FUNCTION_BLOCK "G280M_Code"
TITLE =G280M CHAIN CONVEYOR 9001 KILN 1
//COPYRIGHT:    (C) 2009  BUHLER AG, CH-9240 UZWIL, SWITZERLAND
//
//PRODUCT:      WinCoS_BIW01_09
//
//TITLE:        CHAIN CONVEYOR 9001 KILN 1
//                Machine group control
//                Maschinengruppensteuerung
//
//--------------------------------------------------------------------------------
//
//IDENT:        AUTHOR:             DEPT:                              DATE:
//
//P01_FB380.1.0 K.Renz              CSB41                              08.Jun.2010
//             1st Release
//
//--------------------------------------------------------------------------------
//
//PURPOSE:
//
//MANUAL :
//
//RESTRICTIONS:
//
//--------------------------------------------------------------------------------
AUTHOR : KR
FAMILY : USW
VERSION : 9.9


VAR
  Gr : "GCS7_GrpCtrlSub";	//Standard interface to group
  InOutValue1 : DINT ;	//Data for user
  InOutValue2 : DINT ;	//Data for user
  OutWayConflict : BOOL ;	//Data for user
  OutSelectionOk : BOOL ;	//Data for user
  CmdNewValue : BOOL ;	//Data for user
  CmdNewJob : BOOL ;	//Data for user
  OutCodeOK : BOOL ;	//Data for user
  InEndOfJob : BOOL ;	//Data for user
  staWayOk : BOOL ;	//Data for user
  EdgeStartRelease : BOOL ;	//Data for user
  USW8 : BOOL ;	//Data for user
  USW9 : BOOL ;	//Data for user
  USW10 : BOOL ;	//Data for user
  USW11 : BOOL ;	//Data for user
  USW12 : BOOL ;	//Data for user
  USW13 : BOOL ;	//Data for user
  USW14 : BOOL ;	//Data for user
  USW15 : BOOL ;	//Data for user
  A_3922_BZS04 : "GCS7_E_DigInput";	// DigInpCont
  A_3922_BZS05 : "GCS7_E_DigInput";	// DigInpCont
  A_3922_MXZ01 : "GCS7_E_Motor";	// Motor
  A_3921_MXZ01MA : "A_3921_MXZ01MA_Code";	// Motor+6DI
END_VAR
VAR_TEMP
  tmpEnable : BOOL ;
  tmpFlag : BOOL ;
  tmpCmdNext : BOOL ;
  tmpLocal : BOOL ;
  tmpAspOk : BOOL ;
  tmpHWStop : BOOL ;
  tmpInstanzDBNo : INT ;
END_VAR
BEGIN
NETWORK
TITLE =



NETWORK
TITLE =Read command from group control
//Parameter
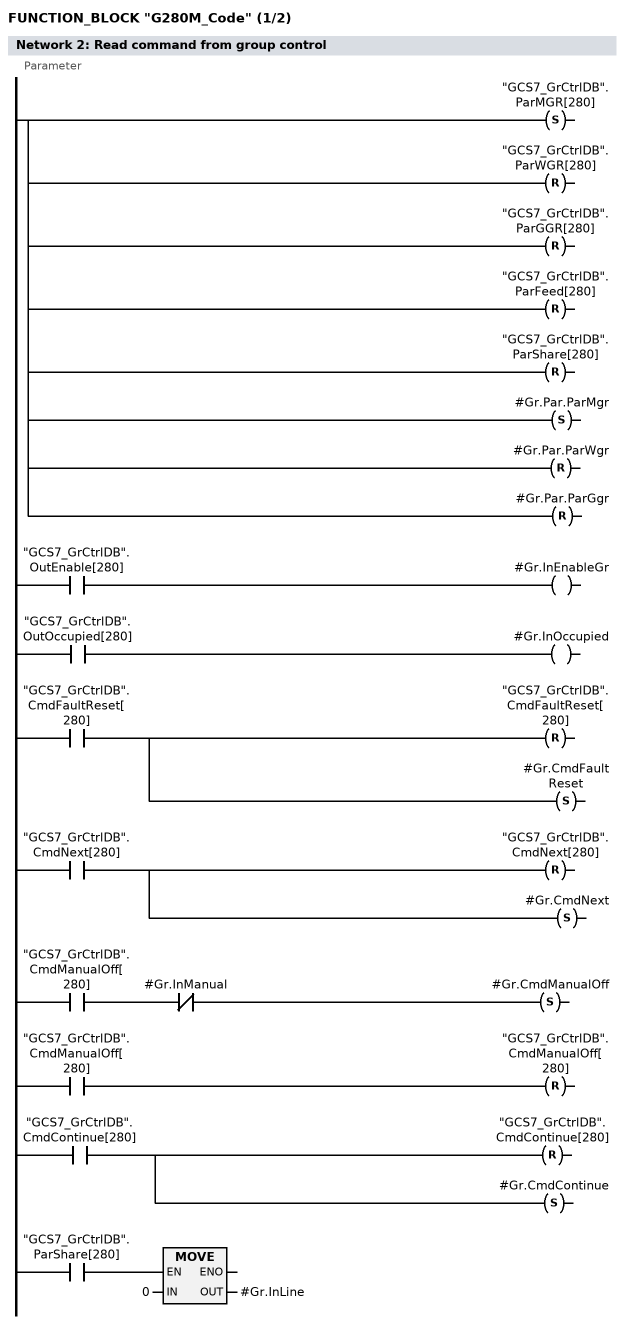
      SET   ;
      S     "GCS7_GrCtrlDB".ParMGR[280];
      R     "GCS7_GrCtrlDB".ParWGR[280];
      R     "GCS7_GrCtrlDB".ParGGR[280];
      R     "GCS7_GrCtrlDB".ParFeed[280];
      R     "GCS7_GrCtrlDB".ParShare[280];
      S     #Gr.Par.ParMgr;
      R     #Gr.Par.ParWgr;
      R     #Gr.Par.ParGgr;
//Command
      U     "GCS7_GrCtrlDB".OutEnable[280];
      =     #Gr.InEnableGr;
      U     "GCS7_GrCtrlDB".OutOccupied[280];
      =     #Gr.InOccupied;
      U     "GCS7_GrCtrlDB".CmdFaultReset[280];
      R     "GCS7_GrCtrlDB".CmdFaultReset[280];
      S     #Gr.CmdFaultReset;
      U     "GCS7_GrCtrlDB".CmdNext[280];
      R     "GCS7_GrCtrlDB".CmdNext[280];
      S     #Gr.CmdNext;

      U     "GCS7_GrCtrlDB".CmdManualOff[280];
      UN    #Gr.InManual;
      S     #Gr.CmdManualOff;
      U     "GCS7_GrCtrlDB".CmdManualOff[280];
      R     "GCS7_GrCtrlDB".CmdManualOff[280];

//      U     "GCS7_GrCtrlDB".CmdManualOff[280]
//      O     "GCS7_GrCtrlDB".OutOccupied[280]
//      R     "GCS7_GrCtrlDB".CmdManualOff[280]
//      S     #Gr.CmdManualOff

      U     "GCS7_GrCtrlDB".CmdContinue[280];
      R     "GCS7_GrCtrlDB".CmdContinue[280];
      S     #Gr.CmdContinue;
//Init Line Number
      U     "GCS7_GrCtrlDB".ParShare[280];
      SPBN  WE00;
      L     0;
      T     #Gr.InLine;
WE00: NOP   0;
NETWORK
TITLE =Call Methode Control
// 1. Handle Interface PCControl
// 2. Prepare mode --> ModePassive,ModeActive,ModeIdling
// 3. Reset global flags of the group
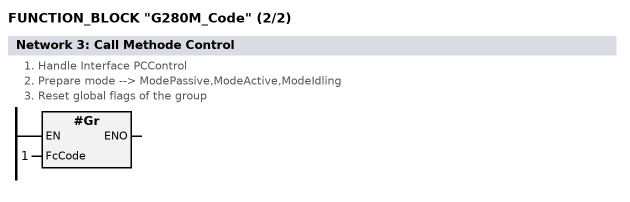
      CALL #Gr (
           FcCode                   := 1);
NETWORK
TITLE =Restart Idling Time

      L     #Gr.Par.ParIdling;
      L     2;
      >=I   ;
      SPB   IdTm;
      T     #Gr.Par.ParIdling;
IdTm: NOP   0;
      CLR   ;
      S     #Gr.CmdRestartIdling;
NETWORK
TITLE =Prepare global flags



NETWORK
TITLE =Set Pattern (Target position)



NETWORK
TITLE =Interlocking WayOk



NETWORK
TITLE =Interlocking Autostart
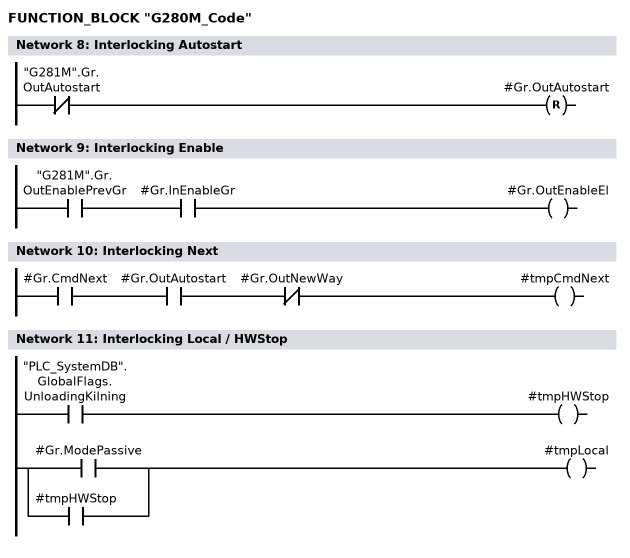

      ON    "G281M".Gr.OutAutostart;
      R     #Gr.OutAutostart;
NETWORK
TITLE =Interlocking Enable

      U     "G281M".Gr.OutEnablePrevGr;
      U     #Gr.InEnableGr;
      =     #Gr.OutEnableEl;

NETWORK
TITLE =Interlocking Next

      U     #Gr.CmdNext;
      U     #Gr.OutAutostart;
      UN    #Gr.OutNewWay;
      =     #tmpCmdNext;

NETWORK
TITLE =Interlocking Local / HWStop

      U     "PLC_SystemDB".GlobalFlags.UnloadingKilning;
      =     #tmpHWStop;

      U     #Gr.ModePassive;
      O     #tmpHWStop;
      =     #tmpLocal;

NETWORK
TITLE =Interlocking Start Warning

      NOP   0;
//- Restart after fault --
      U     #Gr.CmdFaultReset;
      U     #Gr.VarFault;
      S     "SYS_StartWarningDB".Area[10].CmdResetStartWarning;
//- Run Timer --
      AUF   "G280M";
      CALL "GCS7_StartWarning" , "SYS_StartWarningDB" (
           InModeHigher             := FALSE,
           InArea                   := 10,
           InEnable                 := #Gr.OutEnableEl,
           InLocal                  := #tmpLocal,
           InStarted                := #Gr.VarStarted,
           InCmdNext                := #tmpCmdNext,
           OutCmdNext               := #tmpCmdNext,
           OutStartwarning          := #Gr.VarStartwarning);
//- Store Startwarning done  --
//- Reset Autostart --
      U     "SYS_StartWarningDB".TmpArea.OutStartReleaseRunningL;
      FN    #EdgeStartRelease;
      U     #Gr.VarFault;
      R     #Gr.OutAutostart;
NETWORK
TITLE ==A-3922-BZS04 : OUTLET FLAP CLOSED

      NOP   0;
//-InLocal---
      U     #tmpLocal;
      =     #A_3922_BZS04.InLocal;
//
//-Monitoring---
      CLR   ;
      =     #A_3922_BZS04.InMonTrue;
      CLR   ;
      =     #A_3922_BZS04.InMonFalse;
//
//-PreAlarm---
      CLR   ;
      =     #A_3922_BZS04.InPreAlarmTrue;
      CLR   ;
      =     #A_3922_BZS04.InPreAlarmFalse;
//
//-Additional commands---
//      CLR
//      S     #A_3922_BZS04.CmdRunTimeOutTime
//
//-Read inputs---
      U     "A_3922_BZS04_I1";
      =     #A_3922_BZS04.InpTrue;
      U     "PLC_SystemDB".GlobalFlags.UnloadingKilning;
      =     #A_3922_BZS04.InHWStop;
      U     "PLC_DPInfo".Master[1].SlavesError[114];
      =     #A_3922_BZS04.InDPFault;
//
//-Set Parameters---
//
//-Call object control---
      CALL #A_3922_BZS04 ;
//
//-Write outputs---
NETWORK
TITLE ==A-3922-BZS05 : OUTLET FLAP OPENED

      NOP   0;
//-InLocal---
      U     #tmpLocal;
      =     #A_3922_BZS05.InLocal;
//
//-Monitoring---
      CLR   ;
      =     #A_3922_BZS05.InMonTrue;
      CLR   ;
      =     #A_3922_BZS05.InMonFalse;
//
//-PreAlarm---
      CLR   ;
      =     #A_3922_BZS05.InPreAlarmTrue;
      CLR   ;
      =     #A_3922_BZS05.InPreAlarmFalse;
//
//-Additional commands---
//      CLR
//      S     #A_3922_BZS05.CmdRunTimeOutTime
//
//-Read inputs---
      U     "A_3922_BZS05_I1";
      =     #A_3922_BZS05.InpTrue;
      U     "PLC_SystemDB".GlobalFlags.UnloadingKilning;
      =     #A_3922_BZS05.InHWStop;
      U     "PLC_DPInfo".Master[1].SlavesError[114];
      =     #A_3922_BZS05.InDPFault;
//
//-Set Parameters---
//
//-Call object control---
      CALL #A_3922_BZS05 ;
//
//-Write outputs---
NETWORK
TITLE ==A-3922-MXZ01 : OUTLET FLAP DRIVE CLOSE
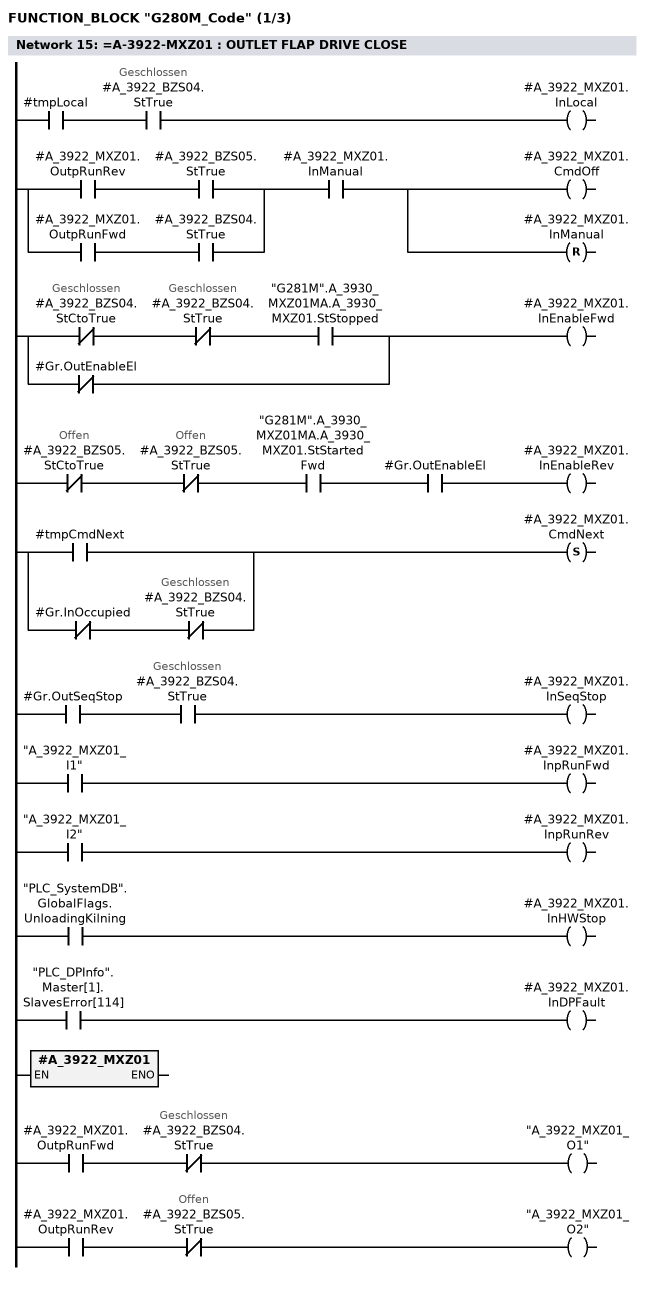

      NOP   0;
//-InLocal---
      U     #tmpLocal;
      U(    ;
      O     #A_3922_BZS04.StTrue; // Geschlossen
//      O     #A_3922_BZS05.StTrue        // Offen
      )     ;
      =     #A_3922_MXZ01.InLocal;
//
//-Interlocking manual---
      U(    ;
      U     #A_3922_MXZ01.OutpRunRev;
      U     #A_3922_BZS05.StTrue;
      O     ;
      U     #A_3922_MXZ01.OutpRunFwd;
      U     #A_3922_BZS04.StTrue;
      )     ;
      U     #A_3922_MXZ01.InManual;
      =     #A_3922_MXZ01.CmdOff;
      R     #A_3922_MXZ01.InManual;
//      S     #A_3922_MXZ01.CmdFaultReset

//-Interlocking---
      UN    #A_3922_BZS04.StCtoTrue; // Geschlossen
      UN    #A_3922_BZS04.StTrue; // Geschlossen
      U     "G281M".A_3930_MXZ01MA.A_3930_MXZ01.StStopped;
      ON    #Gr.OutEnableEl;
      =     #A_3922_MXZ01.InEnableFwd;

      UN    #A_3922_BZS05.StCtoTrue; // Offen
      UN    #A_3922_BZS05.StTrue; // Offen
      U     "G281M".A_3930_MXZ01MA.A_3930_MXZ01.StStartedFwd;
      U     #Gr.OutEnableEl;
      =     #A_3922_MXZ01.InEnableRev;
//
      U     #tmpCmdNext;
      O(    ;
      UN    #Gr.InOccupied;
      UN    #A_3922_BZS04.StTrue; // Geschlossen
      )     ;
      S     #A_3922_MXZ01.CmdNext;
//
      U     #Gr.OutSeqStop;
      U     #A_3922_BZS04.StTrue; // Geschlossen
      =     #A_3922_MXZ01.InSeqStop;
//
//-Read inputs---
      U     "A_3922_MXZ01_I1";
      =     #A_3922_MXZ01.InpRunFwd;
      U     "A_3922_MXZ01_I2";
      =     #A_3922_MXZ01.InpRunRev;
      U     "PLC_SystemDB".GlobalFlags.UnloadingKilning;
      =     #A_3922_MXZ01.InHWStop;
      U     "PLC_DPInfo".Master[1].SlavesError[114];
      =     #A_3922_MXZ01.InDPFault;
//
//-Set Parameters---
//
//-Call object control---
      CALL #A_3922_MXZ01 ;
//
//-Write outputs---
      U     #A_3922_MXZ01.OutpRunFwd;
      UN    #A_3922_BZS04.StTrue; // Geschlossen
      =     "A_3922_MXZ01_O1";
      U     #A_3922_MXZ01.OutpRunRev;
      UN    #A_3922_BZS05.StTrue; // Offen
      =     "A_3922_MXZ01_O2";
NETWORK
TITLE ==A-3921-MXZ01MA : CHAIN CONVEYOR UNDER KILN 1
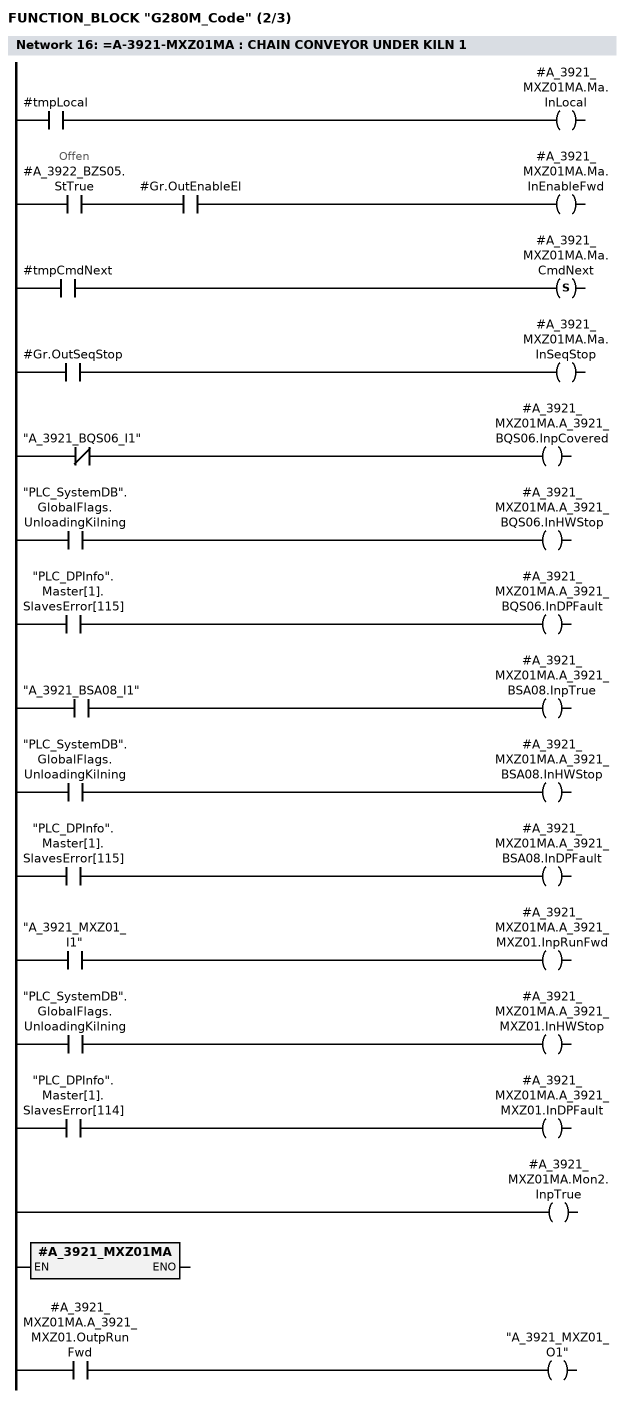

      NOP   0;
//-InLocal---
      U     #tmpLocal;
      =     #A_3921_MXZ01MA.Ma.InLocal;
//
//-Interlocking---
      U     #A_3922_BZS05.StTrue; // Offen
      U     #Gr.OutEnableEl;
      =     #A_3921_MXZ01MA.Ma.InEnableFwd;
//
      U     #tmpCmdNext;
      S     #A_3921_MXZ01MA.Ma.CmdNext;
//
      U     #Gr.OutSeqStop;
      =     #A_3921_MXZ01MA.Ma.InSeqStop;
//
//=Values and commands of elements===
//-=A-3921-BQS06---
//      CLR
//      S     #A_3921_MXZ01MA.A_3921_BQS06.CmdRunTimeOutTime
//-=A-3921-BSA08---
//      CLR
//      S     #A_3921_MXZ01MA.A_3921_BSA08.CmdRunTimeOutTime
//
//-Read inputs of elements---
      UN    "A_3921_BQS06_I1";
      =     #A_3921_MXZ01MA.A_3921_BQS06.InpCovered;
      U     "PLC_SystemDB".GlobalFlags.UnloadingKilning;
      =     #A_3921_MXZ01MA.A_3921_BQS06.InHWStop;
      U     "PLC_DPInfo".Master[1].SlavesError[115];
      =     #A_3921_MXZ01MA.A_3921_BQS06.InDPFault;
      U     "A_3921_BSA08_I1";
      =     #A_3921_MXZ01MA.A_3921_BSA08.InpTrue;
      U     "PLC_SystemDB".GlobalFlags.UnloadingKilning;
      =     #A_3921_MXZ01MA.A_3921_BSA08.InHWStop;
      U     "PLC_DPInfo".Master[1].SlavesError[115];
      =     #A_3921_MXZ01MA.A_3921_BSA08.InDPFault;
      U     "A_3921_MXZ01_I1";
      =     #A_3921_MXZ01MA.A_3921_MXZ01.InpRunFwd;
      U     "PLC_SystemDB".GlobalFlags.UnloadingKilning;
      =     #A_3921_MXZ01MA.A_3921_MXZ01.InHWStop;
      U     "PLC_DPInfo".Master[1].SlavesError[114];
      =     #A_3921_MXZ01MA.A_3921_MXZ01.InDPFault;
      SET   ;
      =     #A_3921_MXZ01MA.Mon2.InpTrue;
//
//-Set Parameters---
//
//-Call object control---
      CALL #A_3921_MXZ01MA ;
//
//-Write outputs---
      U     #A_3921_MXZ01MA.A_3921_MXZ01.OutpRunFwd;
      =     "A_3921_MXZ01_O1";
NETWORK
TITLE =Test Fault
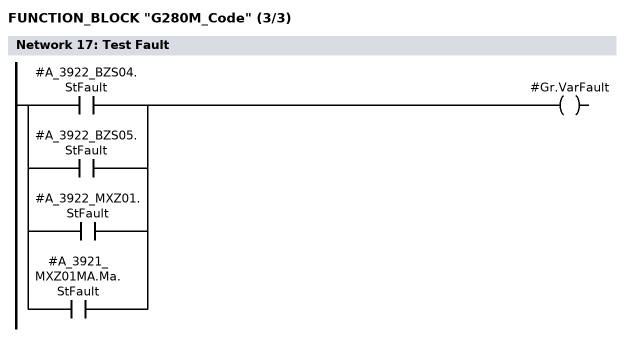

      U     #A_3922_BZS04.StFault;
      O     #A_3922_BZS05.StFault;
      O     #A_3922_MXZ01.StFault;
      O     #A_3921_MXZ01MA.Ma.StFault;
      =     #Gr.VarFault;
NETWORK
TITLE =Test Warning

      CLR   ;
      =     #Gr.OutWarning;
NETWORK
TITLE =Test Stopped
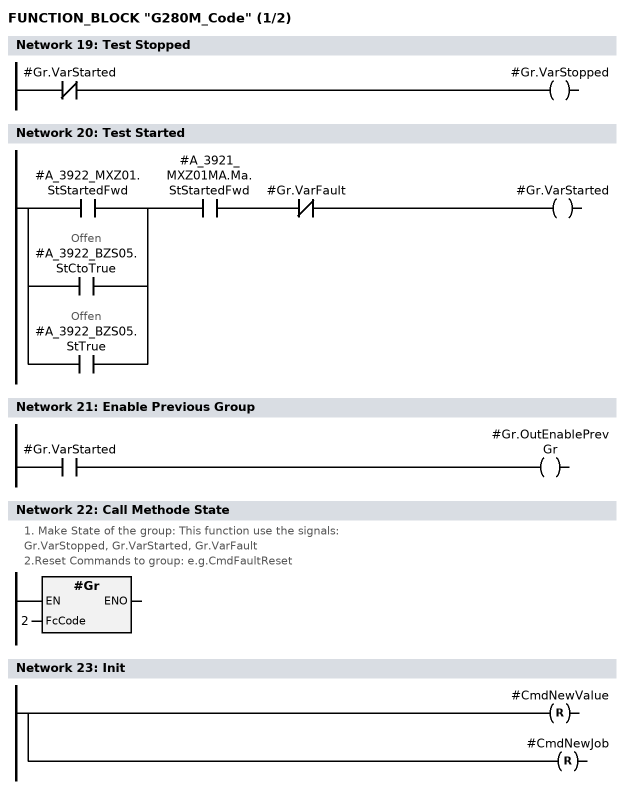

//      U     #A_3922_MXZ01.StStopped
//      U     #A_3921_MXZ01MA.Ma.StStopped
//      UN    #Gr.VarFault
      UN    #Gr.VarStarted;
      =     #Gr.VarStopped;
NETWORK
TITLE =Test Started

      U(    ;
      O     #A_3922_MXZ01.StStartedFwd;
//      O     #A_3922_MXZ01.StStartedRev
      O     #A_3922_BZS05.StCtoTrue; // Offen
      O     #A_3922_BZS05.StTrue; // Offen
      )     ;
      U     #A_3921_MXZ01MA.Ma.StStartedFwd;
//      UN    #Gr.VarStopped
      UN    #Gr.VarFault;
      =     #Gr.VarStarted;
NETWORK
TITLE =Enable Previous Group

      U     #Gr.VarStarted;
      =     #Gr.OutEnablePrevGr;
NETWORK
TITLE =Call Methode State
//1. Make State of the group: This function use the signals:
//        Gr.VarStopped, Gr.VarStarted, Gr.VarFault
//2.Reset Commands to group: e.g.CmdFaultReset
      CALL #Gr (
           FcCode                   := 2);
NETWORK
TITLE =Init

      SET   ;
      R     #CmdNewValue;
      R     #CmdNewJob;
NETWORK
TITLE =Write data to group control
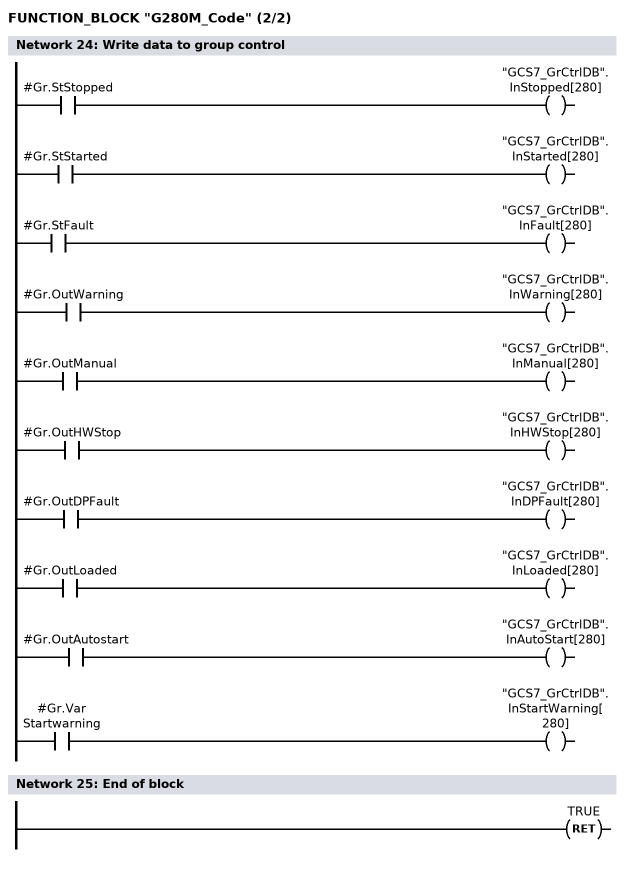

      U     #Gr.StStopped;
      =     "GCS7_GrCtrlDB".InStopped[280];
      U     #Gr.StStarted;
      =     "GCS7_GrCtrlDB".InStarted[280];
      U     #Gr.StFault;
      =     "GCS7_GrCtrlDB".InFault[280];
      U     #Gr.OutWarning;
      =     "GCS7_GrCtrlDB".InWarning[280];
      U     #Gr.OutManual;
      =     "GCS7_GrCtrlDB".InManual[280];
      U     #Gr.OutHWStop;
      =     "GCS7_GrCtrlDB".InHWStop[280];
      U     #Gr.OutDPFault;
      =     "GCS7_GrCtrlDB".InDPFault[280];
      U     #Gr.OutLoaded;
      =     "GCS7_GrCtrlDB".InLoaded[280];
      U     #Gr.OutAutostart;
      =     "GCS7_GrCtrlDB".InAutoStart[280];
      U     #Gr.VarStartwarning;
      =     "GCS7_GrCtrlDB".InStartWarning[280];
NETWORK
TITLE =End of block

      BE    ;

END_FUNCTION_BLOCK

